FUNCTION_BLOCK AB2_B_TO_BYTE (* Composite FB for convert AB2 to BYTE *)
  (* Standard: 61499-2; Description: Copyright (c) 2024 HR Agrartechnik GmbH This program and the accompanying materials are made available under the terms of the Eclipse Public License 2.0 which is available at https://www.eclipse.org/legal/epl-2.0/ SPDX-License-Identifier: EPL-2.0 *)
  (* Version 1.0, 2024-04-24, Franz Höpfinger, HR Agrartechnik GmbH *)
  PACKAGE adapter::conversion::bidirectional;
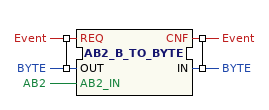
  EVENT_INPUT
    REQ WITH OUT; (* Request to Adapter *)
  END_EVENT
  EVENT_OUTPUT
    CNF WITH IN; (* Confirmation from Adapter *)
  END_EVENT
  VAR_INPUT
    OUT : BYTE; (* Output data to Adapter *)
  END_VAR
  VAR_OUTPUT
    IN : BYTE; (* Input data from Adapter *)
  END_VAR
  SOCKETS
    AB2_IN : adapter::types::bidirectional::AB2; (* Adapter Input *)
  END_SOCKETS
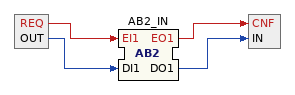
  EVENT_CONNECTIONS
    AB2_IN.EO1 TO CNF;
    REQ TO AB2_IN.EI1;
  END_CONNECTIONS
  DATA_CONNECTIONS
    AB2_IN.DO1 TO IN;
    OUT TO AB2_IN.DI1;
  END_CONNECTIONS
END_FUNCTION_BLOCK
